(* IEC 61131-3 sources: repolevel_ST_code_completion/output/0127完整版本_带planner/repoeval_Decorator_Application/readful_result_no_provide, 7 files *)

(* ---- ConcreteComponment.st ---- *)
VAR
  // Internal variables for description and value
  sDescription : STRING := ''; // Holds the description
  rValue : REAL := 0.0;        // Holds the value
END_VAR

METHOD SetDescription : BOOL
VAR_INPUT
newDescription : STRING;  // Input: New description value
END_VAR
// Correctly assign new description to the internal variable
sDescription := newDescription;
SetDescription := TRUE;   // Return TRUE for success
END_METHOD

METHOD SetValue : BOOL
VAR_INPUT
newValue : REAL;   // Input: New value
END_VAR
// Properly assign new value to the existing internal variable
rValue := newValue;
SetValue := TRUE;   // Return TRUE for success
END_METHOD

METHOD GetInfo : STRING
VAR
combinedInfo : STRING;  // Temporary string for combined output
END_VAR
// Correctly concatenate description and value
combinedInfo := CONCAT(CONCAT(sDescription, ' - '), REAL_TO_STRING(rValue));
GetInfo := combinedInfo;  // Return the combined string
END_METHOD

METHOD InterfaceMethod : BOOL
// Properly return TRUE as confirmation of compatibility with Component_Interface
InterfaceMethod := TRUE;
END_METHOD
END_FUNCTION_BLOCK

(* ---- ConcreteComponment_getDescription.st ---- *)
VAR
    isInitialized : BOOL;
    description : STRING;
END_VAR

IF NOT isInitialized THEN
    RETURN ''; // Return an empty string if the object is not initialized
END_IF;

description := CONCAT('Object Description: ', THIS^.sDescription);
RETURN description;
END_OTHER

(* ---- ConcreteComponment_getValue.st ---- *)
VAR
    rPlainValue : REAL; // Local variable to store the plain value
END_VAR

rPlainValue := THIS^.rValue; // Extract the core value of the object
getValue := rPlainValue; // Assign the extracted value to the return value
RETURN; // Return the result to the caller
END_OTHER

(* ---- ConcreteDecoratorA.st ---- *)
<UNFIXABLE>
VAR_OUTPUT
END_VAR
VAR
	bIsValidComponent : BOOL;
END_VAR

IF tempInputComponent <> 0 THEN
	bIsValidComponent := TRUE;
ELSE
	bIsValidComponent := FALSE;
	RETURN;
END_IF

// Initialize the base class logic
tempComponent := tempInputComponent;

// Execute the core logic of the base component
tempComponent^.Execute();

// Add additional functionality specific to ConcreteDecoratorA
sDescription := CONCAT(tempComponent^.sDescription, ' + DecoratorA');
rValue := tempComponent^.rValue + 10.0;

// Return the updated state or result
RETURN;
END_FUNCTION_BLOCK

(* ---- ConcreteDecoratorA_getDescription.st ---- *)
VAR
    originalDescription : STRING; // Local variable to store the original description
    decoratorDescription : STRING; // Local variable to store the decorator's additional description
    finalDescription : STRING; // Local variable to store the final decorated description
END_VAR

// Step 1: Retrieve the original description of the component
originalDescription := tempInputComponent.getDescription();

// Step 2: Define the decorator's additional description
decoratorDescription := ' - Decorated by A';

// Step 3: Concatenate the original description with the decorator's additional description
finalDescription := CONCAT(originalDescription, decoratorDescription);

// Step 4: Return the final decorated description
getDescription := finalDescription;
END_OTHER

(* ---- ConcreteDecoratorA_getValue.st ---- *)
VAR
	// Variable to store the original value of the component
	rOriginalValue : REAL;
	// Variable to store the fixed decoration value
	rDecorationValue : REAL := 0.5;
END_VAR

// Step 1: Get the original value from the component
rOriginalValue := tempInputComponent.getValue();

// Step 2: Add the fixed decoration value
getValue := rOriginalValue + rDecorationValue;

// Step 3: Return the new value
RETURN;
END_OTHER

(* ---- ConcreteDecoratorC.st ---- *)
VAR
    // Local variable to store the enhanced description
    sEnhancedDescription : STRING;
    // Local variable to store the enhanced value
    rEnhancedValue : REAL;
END_VAR

tempComponent := tempInputComponent; // Step 1: Pass the reference to the parent class

sDescription := tempComponent.sDescription; // Step 2: Execute existing functionality
rValue := tempComponent.rValue;

sEnhancedDescription := CONCAT(sDescription, ' - Enhanced by ConcreteDecoratorC'); // Step 3: Add specific enhancement
rEnhancedValue := rValue * 1.1; // Example of extending functionality by modifying the value

sDescription := sEnhancedDescription; // Step 4: Update the description with enhanced value
rValue := rEnhancedValue; // Update the value with enhanced value
END_FUNCTION_BLOCK
